// TIA Portal V20 export
DATA_BLOCK "instPFEBackbone"   // DB253
AUTHOR : DI FA SUP
FAMILY : LPFE
// stored: InstanceOfName LPFE_PFEBackbone, InstanceOfType FB, Namespace PFE
"LPFE_PFEBackbone"
   // VAR_INPUT
   //    plcInfo { ExternalAccessible := 'False'; ExternalVisible := 'False'; ExternalWritable := 'False'} : "LPFE_typePLCInfo";
   //    channelConfigurationTxn { ExternalAccessible := 'False'; ExternalVisible := 'False'; ExternalWritable := 'False'} : "LPFE_typeOutboundChannelConfig";
   //    channelConfigurationToHost { ExternalAccessible := 'False'; ExternalVisible := 'False'; ExternalWritable := 'False'} : Array[0.."LE_NUMBER_OF_INTERFACE_BUFFERS"] of "LPFE_typeRequestChannelConfig";
   //    channelConfigurationMQTTToHost : "LPFE_typeRequestChannelConfigMQTT";
   //    globalRetryConfiguration { ExternalAccessible := 'False'; ExternalVisible := 'False'; ExternalWritable := 'False'} : "LPFE_typeMsgRetryConfig";
   //    blockingMainBufferTime { ExternalAccessible := 'False'; ExternalVisible := 'False'; ExternalWritable := 'False'} : Time;
   //    programName { ExternalAccessible := 'False'; ExternalVisible := 'False'; ExternalWritable := 'False'} : Array[0..15] of Char;
   //    newShiftInitialization { ExternalAccessible := 'False'; ExternalVisible := 'False'; ExternalWritable := 'False'} : Bool;
   // END_VAR
   // VAR_OUTPUT
   //    currentShiftElapsedTime { ExternalWritable := 'False'} : Time;
   // END_VAR
   // VAR_IN_OUT
   //    resourcesSent { ExternalAccessible := 'False'; ExternalVisible := 'False'; ExternalWritable := 'False'} : Bool;
   //    sendResourceEvents { ExternalAccessible := 'False'; ExternalVisible := 'False'; ExternalWritable := 'False'} : Bool;
   //    resetReceived { ExternalAccessible := 'False'; ExternalVisible := 'False'; ExternalWritable := 'False'} : Bool;
   //    mainBufferBlocked { ExternalAccessible := 'False'; ExternalVisible := 'False'; ExternalWritable := 'False'} : Bool;
   //    cleanupAll { ExternalAccessible := 'False'; ExternalVisible := 'False'; ExternalWritable := 'False'} : Bool;
   //    sessionID { ExternalAccessible := 'False'; ExternalVisible := 'False'; ExternalWritable := 'False'} : UDInt;
   //    globalConnectionParametersFromHost : "LPFE_typeConnectionParameters_1";
   //    globalConnectionParametersToHost : Array[0.."LE_NUMBER_OF_INTERFACE_BUFFERS"] of "LPFE_typeConnectionParameters_1";
   //    globalConnectionParametersTxnChannel : "LPFE_typeConnectionParameters_1";
   //    globalHeartbeatConfiguration : "LPFE_typeHeartbeatConfig";
   //    globalHeartbit { ExternalAccessible := 'False'; ExternalVisible := 'False'; ExternalWritable := 'False'} : Bool;
   //    globalHeartbitDead { ExternalAccessible := 'False'; ExternalVisible := 'False'; ExternalWritable := 'False'} : Bool;
   //    fromHostChannel : "LPFE_typePFEDataInChannel";
   //    toHostInterfaceChannels : Array[0.."LE_NUMBER_OF_INTERFACE_BUFFERS"] of "LPFE_typeRequestChannel";
   //    txnChannel : "LPFE_typePFEDataOutChannel";
   //    prtBuffer : Variant;
   //    prtBufferMgmt : "LPFE_typeMsgBuffer";
   //    FNBuffer : Variant;
   //    FNBufferMgmt : "LPFE_typeMsgBuffer";
   //    TelemetryBuffer : Variant;
   //    TelemetryBufferMgmt : "LPFE_typeMsgBuffer";
   //    recordBuffer : Variant;
   //    recordBufferMgmt : "LPFE_typeMsgBuffer";
   //    mainBuffer : Variant;
   //    mainBufferMgmt : "LPFE_typeMsgBuffer";
   //    ackAndResetBuffer : Variant;
   //    ackAndResetBufferMgmt : "LPFE_typeMsgBuffer";
   //    txnBufferArray : Array[*] of "LPFE_typePFEData";
   //    txnBufferVariant : Variant;
   //    txnBufferMgmt : "LPFE_typeMsgBuffer";
   //    nextInUIdForAckAndReset : "LPFE_typeGlobalSeqMgmt";
   //    nextInUIdFromHostResponse : "LPFE_typeGlobalSeqMgmt";
   //    nextInUIdToHostResponse : "LPFE_typeGlobalSeqMgmt";
   //    nextInUIdToHostPacketIdentifier : "LPFE_typeGlobalSeqMgmt";
   //    nextUIdTxnChannel : "LPFE_typeGlobalSeqMgmt";
   //    newTransactions { ExternalAccessible := 'False'; ExternalVisible := 'False'; ExternalWritable := 'False'} : Int;
   //    criticalRecord : "LPFE_typeCriticalRecEnvelope";
   //    criticalEvent : "LPFE_typeCriticalEventEnvelope";
   //    diagnosticsMonitorDataChannels : Array[0.."LE_NUMBER_OF_INTERFACE_BUFFERS"] of "LPFE_typeDiagnosticMonitorChannel";
   //    monitorTransactions : Array[*] of "LPFE_typePFEData";
   //    performanceMeasurements : Array[*] of "LPFE_typeRequestMeasureBuffer";
   //    healthData : "LPFE_typeMonitorData";
   //    pfeManualReset : Bool;
   // END_VAR
   // VAR
   //    instChannelHandlers { ExternalAccessible := 'False'; ExternalVisible := 'False'; ExternalWritable := 'False'} : "LPFE_ChannelHandlers";
   //    instDistributeMessagesToInterfaces { ExternalAccessible := 'False'; ExternalVisible := 'False'; ExternalWritable := 'False'} : "LPFE_DistributeMsgsToInterfaces";
   //    instCopyMonitorData { ExternalAccessible := 'False'; ExternalVisible := 'False'; ExternalWritable := 'False'} : "LPFE_CopyMonitorData";
   //    instCreateTxnEvents { ExternalAccessible := 'False'; ExternalVisible := 'False'; ExternalWritable := 'False'} : "LPFE_CreateTxnEvents";
   //    instCreateResetEvents { ExternalAccessible := 'False'; ExternalVisible := 'False'; ExternalWritable := 'False'} : "LPFE_CreateResetEvents";
   //    instHealthScreenValueCalculation { ExternalAccessible := 'False'; ExternalVisible := 'False'; ExternalWritable := 'False'} : "LPFE_HealthScreenValueCalculation";
   //    statPlcName { ExternalAccessible := 'False'; ExternalVisible := 'False'; ExternalWritable := 'False'} : Array[0..15] of Char;
   //    statPlcArea { ExternalAccessible := 'False'; ExternalVisible := 'False'; ExternalWritable := 'False'} : Array[0..15] of Char;
   //    statPlcSubArea { ExternalAccessible := 'False'; ExternalVisible := 'False'; ExternalWritable := 'False'} : Array[0..23] of Char;
   //    statInitDone { ExternalAccessible := 'False'; ExternalVisible := 'False'; ExternalWritable := 'False'} : Bool;
   //    statNullChar : Char;
   //    statPLCNameString : String;
   //    statPLCNameWString : WString;
   //    statTopicPrefix : WString;
   //    statTopicSuffix : WString;
   //    statUnderscore : WString;
   //    statHostInitializing : Bool;
   //    statNewIPAck { ExternalAccessible := 'False'; ExternalVisible := 'False'; ExternalWritable := 'False'} : Bool;
   // END_VAR
BEGIN
END_DATA_BLOCK
